FUNCTION_BLOCK PUBLIC FB_RGB_LED
VAR_IN_OUT
	Hardware : TYP_RGB_LED_HW;
END_VAR
VAR_INPUT
END_VAR
VAR_OUTPUT
END_VAR
VAR
END_VAR

METHOD PUBLIC SetRGB : REFERENCE TO FB_RGB_LED
VAR_INPUT
	Red : USINT;
	Green : USINT;
	Blue : USINT;
END_VAR
{warning disable C0371}

// Checking the VAR_IN_OUT reference, leave the current method in case of invalid reference
IF NOT __ISVALIDREF(THIS^.Hardware) THEN
     RETURN;
END_IF

THIS^.Hardware.Red.Out.PWM := REAL_TO_INT((USINT_TO_REAL(Red) / 255) * 32767);
THIS^.Hardware.Green.Out.PWM := REAL_TO_INT((USINT_TO_REAL(Green) / 255) * 32767);
THIS^.Hardware.Blue.Out.PWM := REAL_TO_INT((USINT_TO_REAL(Blue) / 255) * 32767);
END_METHOD

END_FUNCTION_BLOCK

(* stored: Version 1.1.0.1, ProductVersion 3.1.4024.12
   POU FB_RGB_LED: Id {74dccedb-5e88-445d-bb93-b267d6d80982}, SpecialFunc None
   Method SetRGB: Id {a38c9d3c-4497-4c2b-bcf4-1b6cccfeebd2} *)
